ABB RobotStudio station: TestingLetters.rsstn

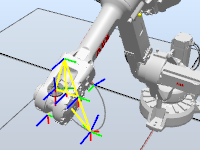
Station TestingLetters (saved by RobotStudio 21.4.9700.0)
Controller IRB2600_12_185
  mechanical unit ROB_1: IRB2600_12_185__02, 6 joints, base frame (0, 0, 0) mm
Layout (positions relative to the parent item):
  - IRB2600_12_185__02 [mechanism, from Robots\IRB2600_12_185_G_02.rslib] at (0, 0, 0) mm; joint values [-0.0485, 0.4593, -0.0093, -0.1903, -1.7519, 0.5651] (rad or m)
  - Part_2 [part], size 0 x 150 x 150 mm
  - Part_3 [part], size 204.9 x 187.3 x 188.4 mm
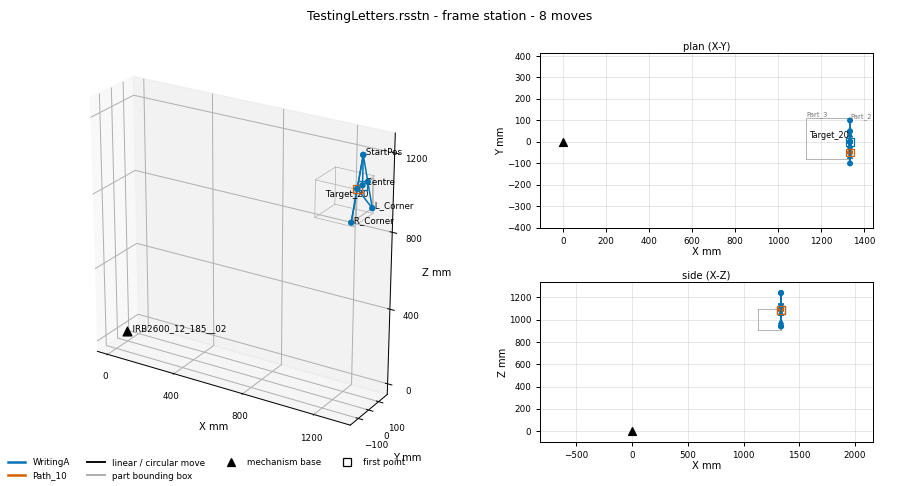
[picture p0: tool path of TestingLetters.rsstn in frame station, 8 of 8 moves have a stored position in this frame; points joined in program order, loops and branches not executed]
Targets, tools, work objects and paths stored in the station, written as RAPID:
! task T_ROB1
MODULE Module1
  CONST robtarget R_Corner:=[[1336.000063563,-100.000004349,940.00009488],[0.706151705,0.00000002,0.70806057,0.000000015],[-1,-1,0,1],[9E+09,9E+09,9E+09,9E+09,9E+09,9E+09]];
  CONST robtarget Centre:=[[1336.000084226,-0.000105515,1089.999909894],[0.706151707,0.000000011,0.708060567,-0.000000006],[-1,-1,0,1],[9E+09,9E+09,9E+09,9E+09,9E+09,9E+09]];
  CONST robtarget L_Corner:=[[1336.000063563,100.000004349,940.00009488],[0.706151705,0.000000006,0.70806057,0.000000011],[0,0,-1,1],[9E+09,9E+09,9E+09,9E+09,9E+09,9E+09]];
  CONST robtarget StartPos:=[[1336.000077935,0,1240.000023955],[0.706151706,0.000000003,0.708060568,0.000000003],[0,0,0,1],[9E+09,9E+09,9E+09,9E+09,9E+09,9E+09]];
  CONST robtarget R_Mid:=[[1336.00007495,-49.999997558,1090.000058219],[0.706151717,0,0.708060557,0.000000002],[-1,-1,0,1],[9E+09,9E+09,9E+09,9E+09,9E+09,9E+09]];
  CONST robtarget L_Mid:=[[1336.000079835,49.999830008,1090.000048773],[0.706151708,0.000000001,0.708060566,0],[0,0,-1,1],[9E+09,9E+09,9E+09,9E+09,9E+09,9E+09]];
  CONST robtarget Target_10:=[[1336,100,940],[0.180407894,-0.26458531,0.050458418,0.945992364],[0,0,0,0],[9E+09,9E+09,9E+09,9E+09,9E+09,9E+09]];
  CONST robtarget Target_20:=[[1131.146597498,-0.535735061,989.137836506],[0.652828066,-0.271690111,-0.271690111,-0.652828066],[0,0,0,0],[9E+09,9E+09,9E+09,9E+09,9E+09,9E+09]];
  CONST robtarget Target_30:=[[1336,-49,1090],[0.946229257,-0.045801741,0.154506016,0.280500063],[0,0,0,0],[9E+09,9E+09,9E+09,9E+09,9E+09,9E+09]];
  PROC WritingA()
    MoveL Centre,v300,fine,tool0\WObj:=wobj0;
    MoveL StartPos,v300,fine,tool0\WObj:=wobj0;
    MoveL R_Corner,v300,fine,tool0\WObj:=wobj0;
    MoveL StartPos,v300,fine,tool0\WObj:=wobj0;
    MoveL L_Corner,v300,fine,tool0\WObj:=wobj0;
    MoveL R_Mid,v300,fine,tool0\WObj:=wobj0;
    MoveL L_Mid,v300,fine,tool0\WObj:=wobj0;
  ENDPROC
  PROC Path_10()
    MoveC Target_20,Target_30,v1000,z100,tool0\WObj:=wobj0;
  ENDPROC
ENDMODULE

